  BlendingMode.EXACT_STOP           : StrReplace('EXACT_STOP ({0})','{0}'           , USINT_TO_STRING(Value));
  BlendingMode.DEFINED_VELOCITY     : StrReplace('DEFINED_VELOCITY ({0})','{0}'     , USINT_TO_STRING(Value));
  BlendingMode.CORNER_DISTANCE      : StrReplace('CORNER_DISTANCE ({0})','{0}'      , USINT_TO_STRING(Value));
  BlendingMode.MAX_CORNER_DEVIATION : StrReplace('MAX_CORNER_DEVIATION ({0})','{0}' , USINT_TO_STRING(Value));
  BlendingMode.CORNER_DISTANCE_2R   : StrReplace('CORNER_DISTANCE_2R ({0})','{0}'   , USINT_TO_STRING(Value));
  BlendingMode.RAMP_OVERLAP         : StrReplace('RAMP_OVERLAP ({0})','{0}'         , USINT_TO_STRING(Value));
  BlendingMode.CORNER_DISTANCE_1R   : StrReplace('CORNER_DISTANCE_1R ({0})','{0}'   , USINT_TO_STRING(Value));

END_CASE

END_FUNCTION

// Library/Functions/Convert/TO_STRING/BYTE_TO_STRING_BIN
FUNCTION BYTE_TO_STRING_BIN : STRING
// ------------------------------------------------------------------------- 
//  SRCI Robot Library                                                
// ------------------------------------------------------------------------- 
//                                                                           
//  Object:      BYTE_TO_STRING_BIN                                       
//  Author:      Thorsten Brach                                                
//  Date:        2025-01-20
//
//  Description:                                              
//    Converts a BYTE to a STRING with binary notation  
//                                                                           
//  Copyright: 
//    (C) 2024 Thorsten Brach. All rights reserved                                                                                                                                            
//             Licensed under the LGPL-3.0 license.
//                                                                           
//  Disclaimer:                                                                           
//    This project is provided without any guarantee and can be used for   
//    private and commercial purposes. Any use is at the user’s 
//    own risk and responsibility.
//
// -------------------------------------------------------------------------
VAR_INPUT
 /// Value to convert
 Value : BYTE; 
END_VAR

BYTE_TO_STRING_BIN := '2#';

IF (Value.7)
THEN
  BYTE_TO_STRING_BIN := CONCAT(BYTE_TO_STRING_BIN, '1');
ELSE
  BYTE_TO_STRING_BIN := CONCAT(BYTE_TO_STRING_BIN, '0');
END_IF

IF (Value.6)
THEN
  BYTE_TO_STRING_BIN := CONCAT(BYTE_TO_STRING_BIN, '1');
ELSE
  BYTE_TO_STRING_BIN := CONCAT(BYTE_TO_STRING_BIN, '0');
END_IF

IF (Value.5)
THEN
  BYTE_TO_STRING_BIN := CONCAT(BYTE_TO_STRING_BIN, '1');
ELSE
  BYTE_TO_STRING_BIN := CONCAT(BYTE_TO_STRING_BIN, '0');
END_IF

IF (Value.4)
THEN
  BYTE_TO_STRING_BIN := CONCAT(BYTE_TO_STRING_BIN, '1_');
ELSE
  BYTE_TO_STRING_BIN := CONCAT(BYTE_TO_STRING_BIN, '0_');
END_IF

IF (Value.3)
THEN
  BYTE_TO_STRING_BIN := CONCAT(BYTE_TO_STRING_BIN, '1');
ELSE
  BYTE_TO_STRING_BIN := CONCAT(BYTE_TO_STRING_BIN, '0');
END_IF

IF (Value.2)
THEN
  BYTE_TO_STRING_BIN := CONCAT(BYTE_TO_STRING_BIN, '1');
ELSE
  BYTE_TO_STRING_BIN := CONCAT(BYTE_TO_STRING_BIN, '0');
END_IF

IF (Value.1)
THEN
  BYTE_TO_STRING_BIN := CONCAT(BYTE_TO_STRING_BIN, '1');
ELSE
  BYTE_TO_STRING_BIN := CONCAT(BYTE_TO_STRING_BIN, '0');
END_IF


IF (Value.0)
THEN
  BYTE_TO_STRING_BIN := CONCAT(BYTE_TO_STRING_BIN, '1');
ELSE
  BYTE_TO_STRING_BIN := CONCAT(BYTE_TO_STRING_BIN, '0');
END_IF


BYTE_TO_STRING_BIN := CONCAT(BYTE_TO_STRING_BIN, ' (');
BYTE_TO_STRING_BIN := CONCAT(BYTE_TO_STRING_BIN, WORD_TO_STRING(Value));
BYTE_TO_STRING_BIN := CONCAT(BYTE_TO_STRING_BIN, ')');

END_FUNCTION

// Library/Functions/Convert/TO_STRING/CIRC_MODE_TO_STRING
FUNCTION CIRC_MODE_TO_STRING : STRING
// ------------------------------------------------------------------------- 
//  SRCI Robot Library                                                
// ------------------------------------------------------------------------- 
//                                                                           
//  Object:      CIRC_MODE_TO_STRING                                       
//  Author:      Thorsten Brach                                                
//  Date:        2025-01-30
//
//  Description:                                              
//   
//                                                                           
//  Copyright: 
//    (C) 2025 Thorsten Brach. All rights reserved                                                                                                                                            
//             Licensed under the LGPL-3.0 license.
//                                                                           
//  Disclaimer:                                                                           
//    This project is provided without any guarantee and can be used for   
//    private and commercial purposes. Any use is at the user’s 
//    own risk and responsibility.
//
// -------------------------------------------------------------------------
VAR_INPUT
  /// CircMode
  Value : CircMode;
END_VAR

CASE Value 
OF

  CircMode.BORDER            : StrReplace('BORDER ({0})'            ,'{0}' , SINT_TO_STRING(Value));
  CircMode.CENTER            : StrReplace('CENTER ({0})'            ,'{0}' , SINT_TO_STRING(Value));
  CircMode.CENTER_WITH_ANGLE : StrReplace('CENTER_WITH_ANGLE ({0})' ,'{0}' , SINT_TO_STRING(Value));
  CircMode.RADIUS            : StrReplace('RADIUS ({0})'            ,'{0}' , SINT_TO_STRING(Value));

END_CASE

END_FUNCTION

// Library/Functions/Convert/TO_STRING/CIRC_PLANE_TO_STRING
FUNCTION CIRC_PLANE_TO_STRING : STRING
// ------------------------------------------------------------------------- 
//  SRCI Robot Library                                                
// ------------------------------------------------------------------------- 
//                                                                           
//  Object:      CIRC_PLANE_TO_STRING                                       
//  Author:      Thorsten Brach                                                
//  Date:        2025-01-30
//
//  Description:                                              
//   
//                                                                           
//  Copyright: 
//    (C) 2025 Thorsten Brach. All rights reserved                                                                                                                                            
//             Licensed under the LGPL-3.0 license.
//                                                                           
//  Disclaimer:                                                                           
//    This project is provided without any guarantee and can be used for   
//    private and commercial purposes. Any use is at the user’s 
//    own risk and responsibility.
//
// -------------------------------------------------------------------------
VAR_INPUT
  /// CircPlane
  Value : CircPlane;
END_VAR

CASE Value 
OF

  CircPlane.XZ_PLANE : StrReplace('XZ_PLANE ({0})' ,'{0}' , SINT_TO_STRING(Value));
  CircPlane.YZ_PLANE : StrReplace('YZ_PLANE ({0})' ,'{0}' , SINT_TO_STRING(Value));
  CircPlane.XY_PLANE : StrReplace('XY_PLANE ({0})' ,'{0}' , SINT_TO_STRING(Value));

END_CASE

END_FUNCTION

// Library/Functions/Convert/TO_STRING/CMD_MESSAGE_STATE_TO_STRING
FUNCTION CMD_MESSAGE_STATE_TO_STRING : STRING
// ------------------------------------------------------------------------- 
//  SRCI Robot Library                                                
// ------------------------------------------------------------------------- 
//                                                                           
//  Object:      CMD_MESSAGE_STATE_TO_STRING                                       
//  Author:      Thorsten Brach                                                
//  Date:        2024-11-16
//
//  Description:                                              
//   
//                                                                           
//  Copyright: 
//    (C) 2024 Thorsten Brach. All rights reserved                                                                                                                                            
//             Licensed under the LGPL-3.0 license.
//                                                                           
//  Disclaimer:                                                                           
//    This project is provided without any guarantee and can be used for   
//    private and commercial purposes. Any use is at the user’s 
//    own risk and responsibility.
//
// -------------------------------------------------------------------------
VAR_INPUT
  /// Command message state
  Value : CmdMessageState;
END_VAR

CASE Value
OF
  CmdMessageState.EMPTY               : CMD_MESSAGE_STATE_TO_STRING := StrReplace('EMPTY ({0})'              ,'{0}', USINT_TO_STRING(Value));
  CmdMessageState.CREATED             : CMD_MESSAGE_STATE_TO_STRING := StrReplace('CREATED ({0})'            ,'{0}', USINT_TO_STRING(Value));
  CmdMessageState.BUFFERED            : CMD_MESSAGE_STATE_TO_STRING := StrReplace('BUFFERED ({0})'           ,'{0}', USINT_TO_STRING(Value));
  CmdMessageState.BUFFERED_IN_PLANNER : CMD_MESSAGE_STATE_TO_STRING := StrReplace('BUFFERED_IN_PLANNER ({0})','{0}', USINT_TO_STRING(Value));
  CmdMessageState.ACTIVE              : CMD_MESSAGE_STATE_TO_STRING := StrReplace('ACTIVE ({0})'             ,'{0}', USINT_TO_STRING(Value));
  CmdMessageState.INTERRUPTED         : CMD_MESSAGE_STATE_TO_STRING := StrReplace('INTERRUPTED ({0})'        ,'{0}', USINT_TO_STRING(Value));
  CmdMessageState.ABORT_REQUEST       : CMD_MESSAGE_STATE_TO_STRING := StrReplace('ABORT_REQUEST ({0})'      ,'{0}', USINT_TO_STRING(Value));
  CmdMessageState.DONE                : CMD_MESSAGE_STATE_TO_STRING := StrReplace('DONE ({0})'               ,'{0}', USINT_TO_STRING(Value));
  CmdMessageState.ABORTED             : CMD_MESSAGE_STATE_TO_STRING := StrReplace('ABORTED ({0})'            ,'{0}', USINT_TO_STRING(Value));
  CmdMessageState.ERROR               : CMD_MESSAGE_STATE_TO_STRING := StrReplace('ERROR ({0})'              ,'{0}', USINT_TO_STRING(Value));
ELSE
  CMD_MESSAGE_STATE_TO_STRING := CONCAT('CmdMessageStateToString-Function: Error -> no parsing for value ', USINT_TO_STRING(Value));
END_CASE

END_FUNCTION

// Library/Functions/Convert/TO_STRING/CMD_TYPE_TO_STRING
FUNCTION CMD_TYPE_TO_STRING : String
// ------------------------------------------------------------------------- 
//  SRCI Robot Library                                                
// ------------------------------------------------------------------------- 
//                                                                           
//  Object:      CMD_TYPE_TO_STRING                                       
//  Author:      Thorsten Brach                                                
//  Date:        2024-11-16
//
//  Description:                                              
//   
//                                                                           
//  Copyright: 
//    (C) 2024 Thorsten Brach. All rights reserved                                                                                                                                            
//             Licensed under the LGPL-3.0 license.
//                                                                           
//  Disclaimer:                                                                           
//    This project is provided without any guarantee and can be used for   
//    private and commercial purposes. Any use is at the user’s 
//    own risk and responsibility.
//
// -------------------------------------------------------------------------
VAR_INPUT
  /// command type
  Value : CmdType;
END_VAR

CASE Value 
OF
  CmdType.RobotTask                   : CMD_TYPE_TO_STRING := StrReplace('RobotTask ({0})','{0}'                  , UINT_TO_STRING(CmdType.RobotTask));   

  CmdType.ReadRobotData               : CMD_TYPE_TO_STRING := StrReplace('ReadRobotData ({0})','{0}'              , UINT_TO_STRING(CmdType.ReadRobotData));

  CmdType.EnableRobot                 : CMD_TYPE_TO_STRING := StrReplace('EnableRobot ({0})','{0}'                , UINT_TO_STRING(CmdType.EnableRobot));  

  CmdType.GroupReset                  : CMD_TYPE_TO_STRING := StrReplace('GroupReset ({0})','{0}'                 , UINT_TO_STRING(CmdType.GroupReset));  

  CmdType.ReadActualPosition          : CMD_TYPE_TO_STRING := StrReplace('ReadActualPosition ({0})','{0}'         , UINT_TO_STRING(CmdType.ReadActualPosition));

  CmdType.ReadActualPositionCyclic    : CMD_TYPE_TO_STRING := StrReplace('ReadActualPositionCyclic ({0})','{0}'   , UINT_TO_STRING(CmdType.ReadActualPositionCyclic));  

  CmdType.ReadDHParameter             : CMD_TYPE_TO_STRING := StrReplace('ReadDHParameter ({0})','{0}'            , UINT_TO_STRING(CmdType.ReadDHParameter));  

  CmdType.RestartController           : CMD_TYPE_TO_STRING := StrReplace('RestartController ({0})','{0}'          , UINT_TO_STRING(CmdType.RestartController));  

  CmdType.ReadActualTCPVelocity       : CMD_TYPE_TO_STRING := StrReplace('ReadActualTCPVelocity ({0})','{0}'      , UINT_TO_STRING(CmdType.ReadActualTCPVelocity));  

  CmdType.UserLogin                   : CMD_TYPE_TO_STRING := StrReplace('UserLogin ({0})','{0}'                  , UINT_TO_STRING(CmdType.UserLogin));

  CmdType.SwitchLanguage              : CMD_TYPE_TO_STRING := StrReplace('SwitchLanguage ({0})','{0}'             , UINT_TO_STRING(CmdType.SwitchLanguage));

  CmdType.ExchangeConfiguration       : CMD_TYPE_TO_STRING := StrReplace('ExchangeConfiguration ({0})','{0}'      , UINT_TO_STRING(CmdType.ExchangeConfiguration));

  CmdType.SetSequence                 : CMD_TYPE_TO_STRING := StrReplace('SetSequence ({0})','{0}'                , UINT_TO_STRING(CmdType.SetSequence));

  CmdType.ChangeSpeedOverride         : CMD_TYPE_TO_STRING := StrReplace('ChangeSpeedOverride ({0})','{0}'        , UINT_TO_STRING(CmdType.ChangeSpeedOverride));

  CmdType.ReadMessages                : CMD_TYPE_TO_STRING := StrReplace('ReadMessages ({0})','{0}'               , UINT_TO_STRING(CmdType.ReadMessages));

  CmdType.ReadRobotReferenceDynamics  : CMD_TYPE_TO_STRING := StrReplace('ReadRobotReferenceDynamics ({0})','{0}' , UINT_TO_STRING(CmdType.ReadRobotReferenceDynamics));  

  CmdType.WriteFrameData              : CMD_TYPE_TO_STRING := StrReplace('WriteFrameData ({0})','{0}'             , UINT_TO_STRING(CmdType.WriteFrameData));

  CmdType.WriteToolData               : CMD_TYPE_TO_STRING := StrReplace('WriteToolData ({0})','{0}'              , UINT_TO_STRING(CmdType.WriteToolData));

  CmdType.WriteLoadData               : CMD_TYPE_TO_STRING := StrReplace('WriteLoadData ({0})','{0}'              , UINT_TO_STRING(CmdType.WriteLoadData));

  CmdType.WriteRobotReferenceDynamics : CMD_TYPE_TO_STRING := StrReplace('WriteRobotReferenceDynamics ({0})','{0}', UINT_TO_STRING(CmdType.WriteRobotReferenceDynamics));

  CmdType.WriteRobotDefaultDynamics   : CMD_TYPE_TO_STRING := StrReplace('WriteRobotDefaultDynamics ({0})'  ,'{0}', UINT_TO_STRING(CmdType.WriteRobotDefaultDynamics));

  CmdType.ReadRobotDefaultDynamics    : CMD_TYPE_TO_STRING := StrReplace('ReadRobotDefaultDynamics ({0})'   ,'{0}', UINT_TO_STRING(CmdType.ReadRobotDefaultDynamics));

  CmdType.ReadFrameData               : CMD_TYPE_TO_STRING := StrReplace('ReadFrameData ({0})'              ,'{0}', UINT_TO_STRING(CmdType.ReadFrameData)); 

  CmdType.ReadToolData                : CMD_TYPE_TO_STRING := StrReplace('ReadToolData ({0})','{0}'               , UINT_TO_STRING(CmdType.ReadToolData));

  CmdType.ReadLoadData                : CMD_TYPE_TO_STRING := StrReplace('ReadLoadData ({0})','{0}'               , UINT_TO_STRING(CmdType.ReadLoadData));

  CmdType.ReadRobotSWLimits           : CMD_TYPE_TO_STRING := StrReplace('ReadRobotSWLimits ({0})','{0}'          , UINT_TO_STRING(CmdType.ReadRobotSWLimits));

  CmdType.WriteRobotSWLimits          : CMD_TYPE_TO_STRING := StrReplace('WriteRobotSWLimits ({0})','{0}'         , UINT_TO_STRING(CmdType.WriteRobotSWLimits));

  CmdType.SetOperationMode            : CMD_TYPE_TO_STRING := StrReplace('SetOperationMode ({0})','{0}'           , UINT_TO_STRING(CmdType.SetOperationMode));

  CmdType.ReadWorkArea                : CMD_TYPE_TO_STRING := StrReplace('ReadWorkArea ({0})','{0}'               , UINT_TO_STRING(CmdType.ReadWorkArea));

  CmdType.WriteWorkArea               : CMD_TYPE_TO_STRING := StrReplace('WriteWorkArea ({0})','{0}'              , UINT_TO_STRING(CmdType.WriteWorkArea));

  CmdType.ActivateWorkArea            : CMD_TYPE_TO_STRING := StrReplace('ActivateWorkArea ({0})','{0}'           , UINT_TO_STRING(CmdType.ActivateWorkArea));

  CmdType.MonitorWorkArea             : CMD_TYPE_TO_STRING := StrReplace('MonitorWorkArea ({0})','{0}'            , UINT_TO_STRING(CmdType.MonitorWorkArea));

  CmdType.GroupJog                    : CMD_TYPE_TO_STRING := StrReplace('GroupJog ({0})','{0}'                   , UINT_TO_STRING(CmdType.GroupJog));

  CmdType.MoveLinearAbsolute          : CMD_TYPE_TO_STRING := StrReplace('MoveLinearAbsolute ({0})','{0}'         , UINT_TO_STRING(CmdType.MoveLinearAbsolute));

  CmdType.MoveDirectAbsolute          : CMD_TYPE_TO_STRING := StrReplace('MoveDirectAbsolute ({0})','{0}'         , UINT_TO_STRING(CmdType.MoveDirectAbsolute));

  CmdType.MoveAxesAbsolute            : CMD_TYPE_TO_STRING := StrReplace('MoveAxesAbsolute ({0})','{0}'           , UINT_TO_STRING(CmdType.MoveAxesAbsolute));

  CmdType.GroupStop                   : CMD_TYPE_TO_STRING := StrReplace('GroupStop ({0})','{0}'                  , UINT_TO_STRING(CmdType.GroupStop));

  CmdType.GroupInterrupt              : CMD_TYPE_TO_STRING := StrReplace('GroupInterrupt ({0})','{0}'             , UINT_TO_STRING(CmdType.GroupInterrupt));

  CmdType.GroupContinue               : CMD_TYPE_TO_STRING := StrReplace('GroupContinue ({0})','{0}'              , UINT_TO_STRING(CmdType.GroupContinue));

  CmdType.MoveLinearRelative          : CMD_TYPE_TO_STRING := StrReplace('MoveLinearRelative ({0})','{0}'         , UINT_TO_STRING(CmdType.MoveLinearRelative));

  CmdType.MoveDirectRelative          : CMD_TYPE_TO_STRING := StrReplace('MoveDirectRelative ({0})','{0}'         , UINT_TO_STRING(CmdType.MoveDirectRelative));

  CmdType.MoveAxesRelative            : CMD_TYPE_TO_STRING := StrReplace('MoveAxesRelative ({0})','{0}'           , UINT_TO_STRING(CmdType.MoveAxesRelative));

  CmdType.ReturnToPrimary             : CMD_TYPE_TO_STRING := StrReplace('ReturnToPrimary ({0})','{0}'            , UINT_TO_STRING(CmdType.ReturnToPrimary));

  CmdType.MoveCircularAbsolute        : CMD_TYPE_TO_STRING := StrReplace('MoveCircularAbsolute ({0})','{0}'       , UINT_TO_STRING(CmdType.MoveCircularAbsolute));

  CmdType.MoveCircularRelative        : CMD_TYPE_TO_STRING := StrReplace('MoveCircularRelative ({0})','{0}'       , UINT_TO_STRING(CmdType.MoveCircularRelative));

  CmdType.MoveLinearOffset            : CMD_TYPE_TO_STRING := StrReplace('MoveLinearOffset ({0})','{0}'           , UINT_TO_STRING(CmdType.MoveLinearOffset));

  CmdType.MoveDirectOffset            : CMD_TYPE_TO_STRING := StrReplace('MoveDirectOffset ({0})','{0}'           , UINT_TO_STRING(CmdType.MoveDirectOffset));

  CmdType.WaitTime                    : CMD_TYPE_TO_STRING := StrReplace('WaitTime ({0})','{0}'                   , UINT_TO_STRING(CmdType.WaitTime));

  CmdType.MoveApproachLinear          : CMD_TYPE_TO_STRING := StrReplace('MoveApproachLinear ({0})','{0}'         , UINT_TO_STRING(CmdType.MoveApproachLinear));

  CmdType.MoveDepartLinear            : CMD_TYPE_TO_STRING := StrReplace('MoveDepartLinear ({0})','{0}'           , UINT_TO_STRING(CmdType.MoveDepartLinear));

  CmdType.MoveApproachDirect          : CMD_TYPE_TO_STRING := StrReplace('MoveApproachDirect ({0})','{0}'         , UINT_TO_STRING(CmdType.MoveApproachDirect));

  CmdType.MoveDepartDirect            : CMD_TYPE_TO_STRING := StrReplace('MoveDepartDirect ({0})','{0}'           , UINT_TO_STRING(CmdType.MoveDepartDirect));

  CmdType.SearchHardstop              : CMD_TYPE_TO_STRING := StrReplace('SearchHardstop ({0})','{0}'             , UINT_TO_STRING(CmdType.SearchHardstop));

  CmdType.SearchHardstopJ             : CMD_TYPE_TO_STRING := StrReplace('SearchHardstopJ ({0})','{0}'            , UINT_TO_STRING(CmdType.SearchHardstopJ));

  CmdType.MovePickPlaceLinear         : CMD_TYPE_TO_STRING := StrReplace('MovePickPlaceLinear ({0})','{0}'        , UINT_TO_STRING(CmdType.MovePickPlaceLinear));

  CmdType.MovePickPlaceDirect         : CMD_TYPE_TO_STRING := StrReplace('MovePickPlaceDirect ({0})','{0}'        , UINT_TO_STRING(CmdType.MovePickPlaceDirect));  

  CmdType.ActivateConveyorTracking    : CMD_TYPE_TO_STRING := StrReplace('ActivateConveyorTracking ({0})','{0}'   , UINT_TO_STRING(CmdType.ActivateConveyorTracking));

  CmdType.RedefineTrackingPos         : CMD_TYPE_TO_STRING := StrReplace('RedefineTrackingPos ({0})','{0}'        , UINT_TO_STRING(CmdType.RedefineTrackingPos));

  CmdType.SyncToConveyor              : CMD_TYPE_TO_STRING := StrReplace('SyncToConveyor ({0})','{0}'             , UINT_TO_STRING(CmdType.SyncToConveyor));

  CmdType.ConfigureConveyor           : CMD_TYPE_TO_STRING := StrReplace('ConfigureConveyor ({0})','{0}'          , UINT_TO_STRING(CmdType.ConfigureConveyor));

  CmdType.MoveSuperImposed            : CMD_TYPE_TO_STRING := StrReplace('MoveSuperImposed ({0})','{0}'           , UINT_TO_STRING(CmdType.MoveSuperImposed));

  CmdType.MoveSuperImposedDynamic     : CMD_TYPE_TO_STRING := StrReplace('MoveSuperImposedDynamic ({0})','{0}'    , UINT_TO_STRING(CmdType.MoveSuperImposedDynamic));

  CmdType.ReadDigitalInputs           : CMD_TYPE_TO_STRING := StrReplace('ReadDigitalInputs ({0})','{0}'          , UINT_TO_STRING(CmdType.ReadDigitalInputs));

  CmdType.ReadDigitalOutputs          : CMD_TYPE_TO_STRING := StrReplace('ReadDigitalOutputs ({0})','{0}'         , UINT_TO_STRING(CmdType.ReadDigitalOutputs));

  CmdType.WriteDigitalOutputs         : CMD_TYPE_TO_STRING := StrReplace('WriteDigitalOutputs ({0})','{0}'        , UINT_TO_STRING(CmdType.WriteDigitalOutputs));

  CmdType.ReadIntegers                : CMD_TYPE_TO_STRING := StrReplace('ReadIntegers ({0})','{0}'               , UINT_TO_STRING(CmdType.ReadIntegers));

  CmdType.ReadReals                   : CMD_TYPE_TO_STRING := StrReplace('ReadReals ({0})','{0}'                  , UINT_TO_STRING(CmdType.ReadReals));

  CmdType.WriteIntegers               : CMD_TYPE_TO_STRING := StrReplace('WriteIntegers ({0})','{0}'              , UINT_TO_STRING(CmdType.WriteIntegers));

  CmdType.WriteReals                  : CMD_TYPE_TO_STRING := StrReplace('WriteReals ({0})','{0}'                 , UINT_TO_STRING(CmdType.WriteReals));

  CmdType.MoveLinearCam               : CMD_TYPE_TO_STRING := StrReplace('MoveLinearCam ({0})','{0}'              , UINT_TO_STRING(CmdType.MoveLinearCam));

  CmdType.MoveDirectCam               : CMD_TYPE_TO_STRING := StrReplace('MoveDirectCam ({0})','{0}'              , UINT_TO_STRING(CmdType.MoveDirectCam));

  CmdType.MoveCircularCam             : CMD_TYPE_TO_STRING := StrReplace('MoveCircularCam ({0})','{0}'            , UINT_TO_STRING(CmdType.MoveCircularCam));

  CmdType.ReadAnalogInput             : CMD_TYPE_TO_STRING := StrReplace('ReadAnalogInput ({0})','{0}'            , UINT_TO_STRING(CmdType.ReadAnalogInput));

  CmdType.ReadAnalogOutput            : CMD_TYPE_TO_STRING := StrReplace('ReadAnalogOutput ({0})','{0}'           , UINT_TO_STRING(CmdType.ReadAnalogOutput));

  CmdType.WriteAnalogOutput           : CMD_TYPE_TO_STRING := StrReplace('WriteAnalogOutput ({0})','{0}'          , UINT_TO_STRING(CmdType.WriteAnalogOutput));

  CmdType.MeasuringInput              : CMD_TYPE_TO_STRING := StrReplace('MeasuringInput ({0})','{0}'             , UINT_TO_STRING(CmdType.MeasuringInput));

  CmdType.AbortMeasuringInput         : CMD_TYPE_TO_STRING := StrReplace('AbortMeasuringInput ({0})','{0}'        , UINT_TO_STRING(CmdType.AbortMeasuringInput));

  CmdType.SetTriggerRegister          : CMD_TYPE_TO_STRING := StrReplace('SetTriggerRegister ({0})','{0}'         , UINT_TO_STRING(CmdType.SetTriggerRegister));

  CmdType.SetTriggerLimit             : CMD_TYPE_TO_STRING := StrReplace('SetTriggerLimit ({0})','{0}'            , UINT_TO_STRING(CmdType.SetTriggerLimit));

  CmdType.SetTriggerUser              : CMD_TYPE_TO_STRING := StrReplace('SetTriggerUser ({0})','{0}'             , UINT_TO_STRING(CmdType.SetTriggerUser));

  CmdType.SetTriggerError             : CMD_TYPE_TO_STRING := StrReplace('SetTriggerError ({0})','{0}'            , UINT_TO_STRING(CmdType.SetTriggerError));

  CmdType.ReactAtTrigger              : CMD_TYPE_TO_STRING := StrReplace('ReactAtTrigger ({0})','{0}'             , UINT_TO_STRING(CmdType.ReactAtTrigger));

  CmdType.WaitForTrigger              : CMD_TYPE_TO_STRING := StrReplace('WaitForTrigger ({0})','{0}'             , UINT_TO_STRING(CmdType.WaitForTrigger));

  CmdType.ReadSystemVariable          : CMD_TYPE_TO_STRING := StrReplace('ReadSystemVariable ({0})','{0}'         , UINT_TO_STRING(CmdType.ReadSystemVariable));

  CmdType.WriteSystemVariable         : CMD_TYPE_TO_STRING := StrReplace('WriteSystemVariable ({0})','{0}'        , UINT_TO_STRING(CmdType.WriteSystemVariable));

  CmdType.CalculateForwardKinematic   : CMD_TYPE_TO_STRING := StrReplace('CalculateForwardKinematic ({0})','{0}'  , UINT_TO_STRING(CmdType.CalculateForwardKinematic));

  CmdType.CalculateInverseKinematic   : CMD_TYPE_TO_STRING := StrReplace('CalculateInverseKinematic ({0})','{0}'  , UINT_TO_STRING(CmdType.CalculateInverseKinematic));

  CmdType.CalculateCartesianPosition  : CMD_TYPE_TO_STRING := StrReplace('CalculateCartesianPosition ({0})','{0}' , UINT_TO_STRING(CmdType.CalculateCartesianPosition));

  CmdType.CalculateTool               : CMD_TYPE_TO_STRING := StrReplace('CalculateTool ({0})','{0}'              , UINT_TO_STRING(CmdType.CalculateTool));

  CmdType.CalculateFrame              : CMD_TYPE_TO_STRING := StrReplace('CalculateFrame ({0})','{0}'             , UINT_TO_STRING(CmdType.CalculateFrame));

  CmdType.ActivateNextCommand         : CMD_TYPE_TO_STRING := StrReplace('ActivateNextCommand ({0})','{0}'        , UINT_TO_STRING(CmdType.ActivateNextCommand));

  CmdType.ShiftPosition               : CMD_TYPE_TO_STRING := StrReplace('ShiftPosition ({0})','{0}'              , UINT_TO_STRING(CmdType.ShiftPosition));

  CmdType.SetTriggerMotion            : CMD_TYPE_TO_STRING := StrReplace('SetTriggerMotion ({0})','{0}'           , UINT_TO_STRING(CmdType.SetTriggerMotion));

  CmdType.OpenBrake                   : CMD_TYPE_TO_STRING := StrReplace('OpenBrake ({0})','{0}'                  , UINT_TO_STRING(CmdType.OpenBrake));

  CmdType.CallSubprogram              : CMD_TYPE_TO_STRING := StrReplace('CallSubprogram ({0})','{0}'             , UINT_TO_STRING(CmdType.CallSubprogram));

  CmdType.WriteCallSubprogramCyclic   : CMD_TYPE_TO_STRING := StrReplace('WriteCallSubprogramCyclic ({0})','{0}'  , UINT_TO_STRING(CmdType.WriteCallSubprogramCyclic));

  CmdType.ReadCallSubprogramCyclic    : CMD_TYPE_TO_STRING := StrReplace('ReadCallSubprogramCyclic ({0})','{0}'   , UINT_TO_STRING(CmdType.ReadCallSubprogramCyclic));

  CmdType.StopSubprogram              : CMD_TYPE_TO_STRING := StrReplace('StopSubprogram ({0})','{0}'             , UINT_TO_STRING(CmdType.StopSubprogram));

  CmdType.PathAccuracyMode            : CMD_TYPE_TO_STRING := StrReplace('PathAccuracyMode ({0})','{0}'           , UINT_TO_STRING(CmdType.PathAccuracyMode));

  CmdType.AvoidSingularity            : CMD_TYPE_TO_STRING := StrReplace('AvoidSingularity ({0})','{0}'           , UINT_TO_STRING(CmdType.AvoidSingularity));

  CmdType.ForceControl                : CMD_TYPE_TO_STRING := StrReplace('ForceControl ({0})','{0}'               , UINT_TO_STRING(CmdType.ForceControl));

  CmdType.ForceLimit                  : CMD_TYPE_TO_STRING := StrReplace('ForceLimit ({0})','{0}'                 , UINT_TO_STRING(CmdType.ForceLimit));

  CmdType.ReadActualForce             : CMD_TYPE_TO_STRING := StrReplace('ReadActualForce ({0})','{0}'            , UINT_TO_STRING(CmdType.ReadActualForce));

  CmdType.BrakeTest                   : CMD_TYPE_TO_STRING := StrReplace('BrakeTest ({0})','{0}'                  , UINT_TO_STRING(CmdType.BrakeTest));

  CmdType.SoftSwitchTCP               : CMD_TYPE_TO_STRING := StrReplace('SoftSwitchTCP ({0})','{0}'              , UINT_TO_STRING(CmdType.SoftSwitchTCP));

  CmdType.CreateSpline                : CMD_TYPE_TO_STRING := StrReplace('CreateSpline ({0})','{0}'               , UINT_TO_STRING(CmdType.CreateSpline));

  CmdType.DeleteSpline                : CMD_TYPE_TO_STRING := StrReplace('DeleteSpline ({0})','{0}'               , UINT_TO_STRING(CmdType.DeleteSpline));

  CmdType.MoveSpline                  : CMD_TYPE_TO_STRING := StrReplace('MoveSpline ({0})','{0}'                 , UINT_TO_STRING(CmdType.MoveSpline));

  CmdType.DynamicSpline               : CMD_TYPE_TO_STRING := StrReplace('DynamicSpline ({0})','{0}'              , UINT_TO_STRING(CmdType.DynamicSpline));

  CmdType.LoadMeasurementAutomatic    : CMD_TYPE_TO_STRING := StrReplace('LoadMeasurementAutomatic ({0})','{0}'   , UINT_TO_STRING(CmdType.LoadMeasurementAutomatic));

  CmdType.LoadMeasurementSequential   : CMD_TYPE_TO_STRING := StrReplace('LoadMeasurementSequential ({0})','{0}'  , UINT_TO_STRING(CmdType.LoadMeasurementSequential));

  CmdType.CollisionDetection          : CMD_TYPE_TO_STRING := StrReplace('CollisionDetection ({0})','{0}'         , UINT_TO_STRING(CmdType.CollisionDetection));

  CmdType.FreeDrive                   : CMD_TYPE_TO_STRING := StrReplace('FreeDrive ({0})','{0}'                  , UINT_TO_STRING(CmdType.FreeDrive)); 

  CmdType.UnitMeasurement             : CMD_TYPE_TO_STRING := StrReplace('UnitMeasurement ({0})','{0}'            , UINT_TO_STRING(CmdType.UnitMeasurement));

ELSE
  CMD_TYPE_TO_STRING := CONCAT('CmdTypeToString-Function: Error -> no parsing for value',UINT_TO_STRING(Value));
END_CASE

END_FUNCTION

// Library/Functions/Convert/TO_STRING/COLLISION_REACTION_MODE_TO_STRING
FUNCTION COLLISION_REACTION_MODE_TO_STRING : STRING
// ------------------------------------------------------------------------- 
//  SRCI Robot Library                                                
// ------------------------------------------------------------------------- 
//                                                                           
//  Object:      COLLISION_REACTION_MODE_TO_STRING                                       
//  Author:      Thorsten Brach                                                
//  Date:        2025-01-24
//
//  Description:                                              
//   
//                                                                           
//  Copyright: 
//    (C) 2025 Thorsten Brach. All rights reserved                                                                                                                                            
//             Licensed under the LGPL-3.0 license.
//                                                                           
//  Disclaimer:                                                                           
//    This project is provided without any guarantee and can be used for   
//    private and commercial purposes. Any use is at the user’s 
//    own risk and responsibility.
//
// -------------------------------------------------------------------------
VAR_INPUT
  /// CollisionReactionMode
  Value : CollisionReactionMode;
END_VAR

CASE Value 
OF

  CollisionReactionMode.REVERSED_MOVEMENT : StrReplace('REVERSED_MOVEMENT ({0})','{0}' , USINT_TO_STRING(Value));
  CollisionReactionMode.STANDING_STILL    : StrReplace('STANDING_STILL ({0})'   ,'{0}' , USINT_TO_STRING(Value));

END_CASE

END_FUNCTION

// Library/Functions/Convert/TO_STRING/CONNECTION_MODE_TO_STRING
FUNCTION CONNECTION_MODE_TO_STRING : STRING
// ------------------------------------------------------------------------- 
//  SRCI Robot Library                                                
// ------------------------------------------------------------------------- 
//                                                                           
//  Object:      CONNECTION_MODE_TO_STRING                                       
//  Author:      Thorsten Brach                                                
//  Date:        2025-02-01
//
//  Description:                                              
//   
//                                                                           
//  Copyright: 
//    (C) 2025 Thorsten Brach. All rights reserved                                                                                                                                            
//             Licensed under the LGPL-3.0 license.
//                                                                           
//  Disclaimer:                                                                           
//    This project is provided without any guarantee and can be used for   
//    private and commercial purposes. Any use is at the user’s 
//    own risk and responsibility.
//
// -------------------------------------------------------------------------
VAR_INPUT
  /// ConnectionMode
  Value : ConnectionMode;
END_VAR

CASE Value 
OF

  ConnectionMode.RC_CONNECTED  : StrReplace('RC_CONNECTED ({0})'  ,'{0}' , SINT_TO_STRING(Value));
  ConnectionMode.PLC_CONNECTED : StrReplace('PLC_CONNECTED ({0})' ,'{0}' , SINT_TO_STRING(Value));

END_CASE

END_FUNCTION

// Library/Functions/Convert/TO_STRING/CONVEYOR_TYPE_TO_STRING
FUNCTION CONVEYOR_TYPE_TO_STRING : STRING
// ------------------------------------------------------------------------- 
//  SRCI Robot Library                                                
// ------------------------------------------------------------------------- 
//                                                                           
//  Object:      CONVEYOR_TYPE_TO_STRING                                       
//  Author:      Thorsten Brach                                                
//  Date:        2025-02-01
//
//  Description:                                              
//   
//                                                                           
//  Copyright: 
//    (C) 2025 Thorsten Brach. All rights reserved                                                                                                                                            
//             Licensed under the LGPL-3.0 license.
//                                                                           
//  Disclaimer:                                                                           
//    This project is provided without any guarantee and can be used for   
//    private and commercial purposes. Any use is at the user’s 
//    own risk and responsibility.
//
// -------------------------------------------------------------------------
VAR_INPUT
  /// ConveyorType
  Value : ConveyorType;
END_VAR

CASE Value 
OF

  ConveyorType.LINEAR_CONVEYOR_TRACKING   : StrReplace('LINEAR_CONVEYOR_TRACKING ({0})'   ,'{0}' , USINT_TO_STRING(Value));
  ConveyorType.CIRCULAR_CONVEYOR_TRACKING : StrReplace('CIRCULAR_CONVEYOR_TRACKING ({0})' ,'{0}' , USINT_TO_STRING(Value));
  
END_CASE

END_FUNCTION

// Library/Functions/Convert/TO_STRING/DATA_ENABLE_SYNC_TO_STRING
FUNCTION DATA_ENABLE_SYNC_TO_STRING : STRING
// ------------------------------------------------------------------------- 
//  SRCI Robot Library                                                
// ------------------------------------------------------------------------- 
//                                                                           
//  Object:      DATA_ENABLE_SYNC_TO_STRING                                       
//  Author:      Thorsten Brach                                                
//  Date:        2025-01-24
//
//  Description:                                              
//   
//                                                                           
//  Copyright: 
//    (C) 2025 Thorsten Brach. All rights reserved                                                                                                                                            
//             Licensed under the LGPL-3.0 license.
//                                                                           
//  Disclaimer:                                                                           
//    This project is provided without any guarantee and can be used for   
//    private and commercial purposes. Any use is at the user’s 
//    own risk and responsibility.
//
// -------------------------------------------------------------------------
VAR_INPUT
  /// DataEnableSync
  Value : DataEnableSync;
END_VAR

VAR
  /// temporary byte
 _tmpByte : BYTE;
END_VAR

_tmpByte.0 := Value.EnableSyncTool;
_tmpByte.1 := Value.EnableSyncFrame;
_tmpByte.2 := Value.EnableSyncLoad;
_tmpByte.3 := Value.EnableSyncWorkArea;
_tmpByte.4 := Value.EnableSyncSWLimits;
_tmpByte.5 := Value.EnableSyncDefaultDynamics;
_tmpByte.6 := Value.EnableSyncReferenceDynamics;
_tmpByte.7 := Value.AllowDynamicBlending;

DATA_ENABLE_SYNC_TO_STRING := BYTE_TO_STRING_BIN(_tmpByte);

END_FUNCTION

// Library/Functions/Convert/TO_STRING/DATA_IN_SYNC_TO_STRING
FUNCTION DATA_IN_SYNC_TO_STRING : STRING
// ------------------------------------------------------------------------- 
//  SRCI Robot Library                                                
// ------------------------------------------------------------------------- 
//                                                                           
//  Object:      DATA_IN_SYNC_TO_STRING                                       
//  Author:      Thorsten Brach                                                
//  Date:        2025-01-24
//
//  Description:                                              
//   
//                                                                           
//  Copyright: 
//    (C) 2025 Thorsten Brach. All rights reserved                                                                                                                                            
//             Licensed under the LGPL-3.0 license.
//                                                                           
//  Disclaimer:                                                                           
//    This project is provided without any guarantee and can be used for   
//    private and commercial purposes. Any use is at the user’s 
//    own risk and responsibility.
//
// -------------------------------------------------------------------------
VAR_INPUT
  /// DataInSync
  Value : DataInSync;
END_VAR

VAR
  /// temporary byte
 _tmpByte : BYTE;
END_VAR

_tmpByte.0 := Value.ToolsInSync;
_tmpByte.1 := Value.FramesInSync;
_tmpByte.2 := Value.LoadsInSync;
_tmpByte.3 := Value.WorkAreasInSync;
_tmpByte.4 := Value.SoftwareLimitsInSync;
_tmpByte.5 := Value.DefaultDynamicsInSync;
_tmpByte.6 := Value.ReferenceDynamicsInSync;
_tmpByte.7 := FALSE;

DATA_IN_SYNC_TO_STRING := BYTE_TO_STRING_BIN(_tmpByte);

END_FUNCTION

// Library/Functions/Convert/TO_STRING/DEFINITION_MODE_TO_STRING
FUNCTION DEFINITION_MODE_TO_STRING : STRING
// ------------------------------------------------------------------------- 
//  SRCI Robot Library                                                
// ------------------------------------------------------------------------- 
//                                                                           
//  Object:      DEFINITION_MODE_TO_STRING                                       
//  Author:      Thorsten Brach                                                
//  Date:        2025-02-01
//
//  Description:                                              
//   
//                                                                           
//  Copyright: 
//    (C) 2025 Thorsten Brach. All rights reserved                                                                                                                                            
//             Licensed under the LGPL-3.0 license.
//                                                                           
//  Disclaimer:                                                                           
//    This project is provided without any guarantee and can be used for   
//    private and commercial purposes. Any use is at the user’s 
//    own risk and responsibility.
//
// -------------------------------------------------------------------------
VAR_INPUT
  /// DefinitionMode
  Value : DefinitionMode;
END_VAR

CASE Value 
OF

  DefinitionMode.CENTER : StrReplace('CENTER ({0})','{0}' , USINT_TO_STRING(Value));
  DefinitionMode.FACE   : StrReplace('FACE ({0})'  ,'{0}' , USINT_TO_STRING(Value));

END_CASE

END_FUNCTION

// Library/Functions/Convert/TO_STRING/DETECTION_MODE_TO_STRING
FUNCTION DETECTION_MODE_TO_STRING : STRING
// ------------------------------------------------------------------------- 
//  SRCI Robot Library                                                
// ------------------------------------------------------------------------- 
//                                                                           
//  Object:      DETECTION_MODE_TO_STRING                                       
//  Author:      Thorsten Brach                                                
//  Date:        2025-02-01
//
//  Description:                                              
//   
//                                                                           
//  Copyright: 
//    (C) 2025 Thorsten Brach. All rights reserved                                                                                                                                            
//             Licensed under the LGPL-3.0 license.
//                                                                           
//  Disclaimer:                                                                           
//    This project is provided without any guarantee and can be used for   
//    private and commercial purposes. Any use is at the user’s 
//    own risk and responsibility.
//
// -------------------------------------------------------------------------
VAR_INPUT
  /// DetectionMode
  Value : DetectionMode;
END_VAR

CASE Value 
OF

  DetectionMode.TORQUE             : StrReplace('TORQUE ({0})'             ,'{0}' , USINT_TO_STRING(Value));
  DetectionMode.FORCE              : StrReplace('FORCE ({0})'              ,'{0}' , USINT_TO_STRING(Value));
  DetectionMode.ELECTRICAL_CURRENT : StrReplace('ELECTRICAL_CURRENT ({0})' ,'{0}' , USINT_TO_STRING(Value));
  DetectionMode.FOLLOWING_ERROR    : StrReplace('FOLLOWING_ERROR ({0})'    ,'{0}' , USINT_TO_STRING(Value));

END_CASE

END_FUNCTION

// Library/Functions/Convert/TO_STRING/ERROR_REACTION_TO_STRING
FUNCTION ERROR_REACTION_TO_STRING : STRING
// ------------------------------------------------------------------------- 
//  SRCI Robot Library                                                
// ------------------------------------------------------------------------- 
//                                                                           
//  Object:      ERROR_REACTION_TO_STRING                                       
//  Author:      Thorsten Brach                                                
//  Date:        2025-02-01
//
//  Description:                                              
//   
//                                                                           
//  Copyright: 
//    (C) 2025 Thorsten Brach. All rights reserved                                                                                                                                            
//             Licensed under the LGPL-3.0 license.
//                                                                           
//  Disclaimer:                                                                           
//    This project is provided without any guarantee and can be used for   
//    private and commercial purposes. Any use is at the user’s 
//    own risk and responsibility.
//
// -------------------------------------------------------------------------
VAR_INPUT
  /// ErrorReaction
  Value : ErrorReaction;
END_VAR

CASE Value 
OF

  ErrorReaction.ABORT_AND_MOVE : StrReplace('ABORT_AND_MOVE ({0})','{0}' , USINT_TO_STRING(Value));
  ErrorReaction.ABORT          : StrReplace('ABORT ({0})'         ,'{0}' , USINT_TO_STRING(Value));
  ErrorReaction.NO_REACTION    : StrReplace('NO_REACTION ({0})'   ,'{0}' , USINT_TO_STRING(Value));

END_CASE

END_FUNCTION

// Library/Functions/Convert/TO_STRING/ERROR_TRIGGER_MODE_TO_STRING
FUNCTION ERROR_TRIGGER_MODE_TO_STRING : STRING
// ------------------------------------------------------------------------- 
//  SRCI Robot Library                                                
// ------------------------------------------------------------------------- 
//                                                                           
//  Object:      ERROR_TRIGGER_MODE_TO_STRING                                       
//  Author:      Thorsten Brach                                                
//  Date:        2025-02-01
//
//  Description:                                              
//   
//                                                                           
//  Copyright: 
//    (C) 2025 Thorsten Brach. All rights reserved                                                                                                                                            
//             Licensed under the LGPL-3.0 license.
//                                                                           
//  Disclaimer:                                                                           
//    This project is provided without any guarantee and can be used for   
//    private and commercial purposes. Any use is at the user’s 
//    own risk and responsibility.
//
// -------------------------------------------------------------------------
VAR_INPUT
  /// ErrorTriggerMode
  Value : ErrorTriggerMode;
END_VAR

CASE Value 
OF

  ErrorTriggerMode.ANY_COMMAND                    : StrReplace('ANY_COMMAND ({0})'                    ,'{0}' , SINT_TO_STRING(Value));
  ErrorTriggerMode.GENERAL_COMMANDS               : StrReplace('GENERAL_COMMANDS ({0})'               ,'{0}' , SINT_TO_STRING(Value));
  ErrorTriggerMode.ADMINISTRATIVE_COMMANDS        : StrReplace('ADMINISTRATIVE_COMMANDS ({0})'        ,'{0}' , SINT_TO_STRING(Value));
  ErrorTriggerMode.MOVE_COMMANDS                  : StrReplace('MOVE_COMMANDS ({0})'                  ,'{0}' , SINT_TO_STRING(Value));
  ErrorTriggerMode.PERIPHERY_COMMANDS             : StrReplace('PERIPHERY_COMMANDS ({0})'             ,'{0}' , SINT_TO_STRING(Value));
  ErrorTriggerMode.EXTENDED_COMMANDS              : StrReplace('EXTENDED_COMMANDS ({0})'              ,'{0}' , SINT_TO_STRING(Value));
  ErrorTriggerMode.SPECIFIC_COMMAND_OR_RI_MESSAGE : StrReplace('SPECIFIC_COMMAND_OR_RI_MESSAGE ({0})' ,'{0}' , SINT_TO_STRING(Value));
  ErrorTriggerMode.SPECIFIC_RC_OR_RA_MESSAGE_CODE : StrReplace('SPECIFIC_RC_OR_RA_MESSAGE_CODE ({0})' ,'{0}' , SINT_TO_STRING(Value));
  ErrorTriggerMode.ANY_RI_MESSAGE_CODE            : StrReplace('ANY_RI_MESSAGE_CODE ({0})'            ,'{0}' , SINT_TO_STRING(Value));
  ErrorTriggerMode.ANY_RC_OR_RA_MESSAGE_CODE      : StrReplace('ANY_RC_OR_RA_MESSAGE_CODE ({0})'      ,'{0}' , SINT_TO_STRING(Value));

END_CASE

END_FUNCTION

// Library/Functions/Convert/TO_STRING/EXECUTION_MODE_TO_STRING
FUNCTION EXECUTION_MODE_TO_STRING : STRING
// ------------------------------------------------------------------------- 
//  SRCI Robot Library                                                
// ------------------------------------------------------------------------- 
//                                                                           
//  Object:      EXECUTION_MODE_TO_STRING                                       
//  Author:      Thorsten Brach                                                
//  Date:        2025-01-20
//
//  Description:                                              
//   
//                                                                           
//  Copyright: 
//    (C) 2024 Thorsten Brach. All rights reserved                                                                                                                                            
//             Licensed under the LGPL-3.0 license.
//                                                                           
//  Disclaimer:                                                                           
//    This project is provided without any guarantee and can be used for   
//    private and commercial purposes. Any use is at the user’s 
//    own risk and responsibility.
//
// -------------------------------------------------------------------------
VAR_INPUT
  /// ExecMode
  Value : ExecutionMode;
END_VAR

CASE Value
OF
  ExecutionMode.SEQUENCE_PRIMARY                 : EXECUTION_MODE_TO_STRING := StrReplace('SEQUENCE_PRIMARY ({0})'                 ,'{0}', USINT_TO_STRING(Value));
  ExecutionMode.SEQUENCE_ABORT_OTHERS_PRIMARY    : EXECUTION_MODE_TO_STRING := StrReplace('SEQUENCE_ABORT_OTHERS_PRIMARY ({0})'    ,'{0}', USINT_TO_STRING(Value));
  ExecutionMode.PARALLEL                         : EXECUTION_MODE_TO_STRING := StrReplace('PARALLEL ({0})'                         ,'{0}', USINT_TO_STRING(Value));
  ExecutionMode.CONTINUOUS                       : EXECUTION_MODE_TO_STRING := StrReplace('CONTINUOUS ({0})'                       ,'{0}', USINT_TO_STRING(Value));
  ExecutionMode.TRIGGER_MULTIPLE                 : EXECUTION_MODE_TO_STRING := StrReplace('TRIGGER_MULTIPLE ({0})'                 ,'{0}', USINT_TO_STRING(Value));
  ExecutionMode.SEQUENCE_SECONDARY               : EXECUTION_MODE_TO_STRING := StrReplace('SEQUENCE_SECONDARY ({0})'               ,'{0}', USINT_TO_STRING(Value));
  ExecutionMode.SEQUENCE_ABORT_OTHERS_SECONDARY  : EXECUTION_MODE_TO_STRING := StrReplace('SEQUENCE_ABORT_OTHERS_SECONDARY ({0})'  ,'{0}', USINT_TO_STRING(Value));
  ExecutionMode.STOP_PARALLEL_CONTINUOUS_TRIGGER : EXECUTION_MODE_TO_STRING := StrReplace('STOP_PARALLEL_CONTINUOUS_TRIGGER ({0})' ,'{0}', USINT_TO_STRING(Value));
ELSE
  EXECUTION_MODE_TO_STRING := 'UNKNOWN';
END_CASE

END_FUNCTION

// Library/Functions/Convert/TO_STRING/FRAGMENT_ACTION_TO_STRING
FUNCTION FRAGMENT_ACTION_TO_STRING : STRING
// ------------------------------------------------------------------------- 
//  SRCI Robot Library                                                
// ------------------------------------------------------------------------- 
//                                                                           
//  Object:      FRAGMENT_ACTION_TO_STRING                                       
//  Author:      Thorsten Brach                                                
//  Date:        2024-11-16
//
//  Description:                                              
//   
//                                                                           
//  Copyright: 
//    (C) 2024 Thorsten Brach. All rights reserved                                                                                                                                            
//             Licensed under the LGPL-3.0 license.
//                                                                           
//  Disclaimer:                                                                           
//    This project is provided without any guarantee and can be used for   
//    private and commercial purposes. Any use is at the user’s 
//    own risk and responsibility.
//
// -------------------------------------------------------------------------
VAR_INPUT
  /// Fragment action
  FragmentAction : BYTE;
END_VAR

IF ( FragmentAction.0 )
THEN
 FRAGMENT_ACTION_TO_STRING := CONCAT(FRAGMENT_ACTION_TO_STRING, ' Complete (Bit 0)');
END_IF

IF ( FragmentAction.1 )
THEN
 FRAGMENT_ACTION_TO_STRING := CONCAT(FRAGMENT_ACTION_TO_STRING, ' Reset (Bit 1)');
END_IF

IF ( FragmentAction.2 )
THEN
 FRAGMENT_ACTION_TO_STRING := CONCAT(FRAGMENT_ACTION_TO_STRING, ' Clear (Bit 2)');
END_IF

END_FUNCTION

// Library/Functions/Convert/TO_STRING/FRAME_CALCULATION_MODE_TO_STRING
FUNCTION FRAME_CALCULATION_MODE_TO_STRING : STRING
// ------------------------------------------------------------------------- 
//  SRCI Robot Library                                                
// ------------------------------------------------------------------------- 
//                                                                           
//  Object:      FRAME_CALCULATION_MODE_TO_STRING                                       
//  Author:      Thorsten Brach                                                
//  Date:        2025-02-01
//
//  Description:                                              
//   
//                                                                           
//  Copyright: 
//    (C) 2025 Thorsten Brach. All rights reserved                                                                                                                                            
//             Licensed under the LGPL-3.0 license.
//                                                                           
//  Disclaimer:                                                                           
//    This project is provided without any guarantee and can be used for   
//    private and commercial purposes. Any use is at the user’s 
//    own risk and responsibility.
//
// -------------------------------------------------------------------------
VAR_INPUT
  /// FrameCalculationMode
  Value : FrameCalculationMode;
END_VAR

CASE Value 
OF

  FrameCalculationMode.THREE_POINT_METHOD : StrReplace('THREE_POINT_METHOD ({0})','{0}' , SINT_TO_STRING(Value));
  FrameCalculationMode.FOUR_POINT_METHOD  : StrReplace('FOUR_POINT_METHOD ({0})' ,'{0}' , SINT_TO_STRING(Value));
  FrameCalculationMode.ONE_POINT_METHOD   : StrReplace('ONE_POINT_METHOD ({0})'  ,'{0}' , SINT_TO_STRING(Value));

END_CASE

END_FUNCTION

// Library/Functions/Convert/TO_STRING/IEC_DATE_TO_STRING
FUNCTION IEC_DATE_TO_STRING : STRING
// ------------------------------------------------------------------------- 
//  SRCI Robot Library                                                
// ------------------------------------------------------------------------- 
//                                                                           
//  Object:      IEC_DATE_TO_STRING                                       
//  Author:      Thorsten Brach                                                
//  Date:        2025-02-01
//
//  Description:                                              
//   
//                                                                           
//  Copyright: 
//    (C) 2025 Thorsten Brach. All rights reserved                                                                                                                                            
//             Licensed under the LGPL-3.0 license.
//                                                                           
//  Disclaimer:                                                                           
//    This project is provided without any guarantee and can be used for   
//    private and commercial purposes. Any use is at the user’s 
//    own risk and responsibility.
//
// -------------------------------------------------------------------------
VAR_INPUT
  /// IEC Date
  Value : IEC_DATE;
END_VAR

VAR
  /// temporary date
 _tmpData : DATE;
END_VAR

IEC_DATE_TO_STRING := DATE_TO_STRING(IEC_DATE_TO_DATE(Value));

END_FUNCTION

// Library/Functions/Convert/TO_STRING/IEC_TIME_TO_STRING
FUNCTION IEC_TIME_TO_STRING : STRING
// ------------------------------------------------------------------------- 
//  SRCI Robot Library                                                
// ------------------------------------------------------------------------- 
//                                                                           
//  Object:      ORI_MODE_TO_STRING                                       
//  Author:      Thorsten Brach                                                
//  Date:        2025-01-24
//
//  Description:                                              
//   
//                                                                           
//  Copyright: 
//    (C) 2025 Thorsten Brach. All rights reserved                                                                                                                                            
//             Licensed under the LGPL-3.0 license.
//                                                                           
//  Disclaimer:                                                                           
//    This project is provided without any guarantee and can be used for   
//    private and commercial purposes. Any use is at the user’s 
//    own risk and responsibility.
//
// -------------------------------------------------------------------------
VAR_INPUT
  /// IEC_TIME
  Value : IEC_TIME;
END_VAR
VAR
  /// temporary date
 _tmpData : DATE;
END_VAR

IEC_TIME_TO_STRING := TOD_TO_STRING(IEC_TIME_TO_TIME(Value));

END_FUNCTION

// Library/Functions/Convert/TO_STRING/ORI_MODE_TO_STRING
FUNCTION ORI_MODE_TO_STRING : STRING
// ------------------------------------------------------------------------- 
//  SRCI Robot Library                                                
// ------------------------------------------------------------------------- 
//                                                                           
//  Object:      ORI_MODE_TO_STRING                                       
//  Author:      Thorsten Brach                                                
//  Date:        2025-01-24
//
//  Description:                                              
//   
//                                                                           
//  Copyright: 
//    (C) 2025 Thorsten Brach. All rights reserved                                                                                                                                            
//             Licensed under the LGPL-3.0 license.
//                                                                           
//  Disclaimer:                                                                           
//    This project is provided without any guarantee and can be used for   
//    private and commercial purposes. Any use is at the user’s 
//    own risk and responsibility.
//
// -------------------------------------------------------------------------
VAR_INPUT
  /// OriMode
  Value : OriMode;
END_VAR

CASE Value 
OF

  OriMode.LINEAR_INTERPOLATED : StrReplace('LINEAR_INTERPOLATED ({0})','{0}' , USINT_TO_STRING(Value));
  OriMode.JOINT_INTERPOLATED  : StrReplace('JOINT_INTERPOLATED ({0})' ,'{0}' , USINT_TO_STRING(Value));
  OriMode.FIX                 : StrReplace('FIX ({0})'                ,'{0}' , USINT_TO_STRING(Value));
  OriMode.PATH                : StrReplace('PATH ({0})'               ,'{0}' , USINT_TO_STRING(Value));

END_CASE

END_FUNCTION

// Library/Functions/Convert/TO_STRING/INTERPOLATION_MODE_TO_STRING
FUNCTION INTERPOLATION_MODE_TO_STRING : STRING
// ------------------------------------------------------------------------- 
//  SRCI Robot Library                                                
// ------------------------------------------------------------------------- 
//                                                                           
//  Object:      INTERPOLATION_MODE_TO_STRING                                       
//  Author:      Thorsten Brach                                                
//  Date:        2025-02-01
//
//  Description:                                              
//   
//                                                                           
//  Copyright: 
//    (C) 2025 Thorsten Brach. All rights reserved                                                                                                                                            
//             Licensed under the LGPL-3.0 license.
//                                                                           
//  Disclaimer:                                                                           
//    This project is provided without any guarantee and can be used for   
//    private and commercial purposes. Any use is at the user’s 
//    own risk and responsibility.
//
// -------------------------------------------------------------------------
VAR_INPUT
  /// InterpolationMode
  Value : InterpolationMode;
END_VAR

CASE Value 
OF

  InterpolationMode.LINEAR_INTERPOLATION : StrReplace('LINEAR_INTERPOLATION ({0})' ,'{0}' , USINT_TO_STRING(Value));
  InterpolationMode.DIRECT_INTERPOLATION : StrReplace('DIRECT_INTERPOLATION ({0})' ,'{0}' , USINT_TO_STRING(Value));

END_CASE

END_FUNCTION

// Library/Functions/Convert/TO_STRING/JOG_MODE_TO_STRING
FUNCTION JOG_MODE_TO_STRING : STRING
// ------------------------------------------------------------------------- 
//  SRCI Robot Library                                                
// ------------------------------------------------------------------------- 
//                                                                           
//  Object:      JOG_MODE_TO_STRING                                       
//  Author:      Thorsten Brach                                                
//  Date:        2025-01-20
//
//  Description:                                              
//   
//                                                                           
//  Copyright: 
//    (C) 2025 Thorsten Brach. All rights reserved                                                                                                                                            
//             Licensed under the LGPL-3.0 license.
//                                                                           
//  Disclaimer:                                                                           
//    This project is provided without any guarantee and can be used for   
//    private and commercial purposes. Any use is at the user’s 
//    own risk and responsibility.
//
// -------------------------------------------------------------------------
VAR_INPUT
  /// JogMode
  Value : JogMode;
END_VAR

CASE Value 
OF
  
  JogMode.JOG_FRAME : JOG_MODE_TO_STRING := StrReplace('JOG_FRAME ({0})','{0}' , USINT_TO_STRING(Value));
  JogMode.JOG_TOOL  : JOG_MODE_TO_STRING := StrReplace('JOG_TOOL ({0})','{0}'  , USINT_TO_STRING(Value));
  JogMode.JOG_AXES  : JOG_MODE_TO_STRING := StrReplace('JOG_AXES ({0})','{0}'  , USINT_TO_STRING(Value));

END_CASE

END_FUNCTION

// Library/Functions/Convert/TO_STRING/LIMIT_MODE_TO_STRING
FUNCTION LIMIT_MODE_TO_STRING : STRING
// ------------------------------------------------------------------------- 
//  SRCI Robot Library                                                
// ------------------------------------------------------------------------- 
//                                                                           
//  Object:      LIMIT_MODE_TO_STRING                                       
//  Author:      Thorsten Brach                                                
//  Date:        2025-01-24
//
//  Description:                                              
//   
//                                                                           
//  Copyright: 
//    (C) 2025 Thorsten Brach. All rights reserved                                                                                                                                            
//             Licensed under the LGPL-3.0 license.
//                                                                           
//  Disclaimer:                                                                           
//    This project is provided without any guarantee and can be used for   
//    private and commercial purposes. Any use is at the user’s 
//    own risk and responsibility.
//
// -------------------------------------------------------------------------
VAR_INPUT
  /// LimitMode
  Value : LimitMode;
END_VAR

CASE Value 
OF

  LimitMode.LIMIT_DEFINED    : StrReplace('LIMIT_DEFINED ({0})'    ,'{0}' , USINT_TO_STRING(Value));
  LimitMode.NO_LIMIT_DEFINED : StrReplace('NO_LIMIT_DEFINED ({0})' ,'{0}' , USINT_TO_STRING(Value));

END_CASE

END_FUNCTION

// Library/Functions/Convert/TO_STRING/LOAD_MEASUREMENT_MODE_TO_STRING
FUNCTION LOAD_MEASUREMENT_MODE_TO_STRING : STRING
// ------------------------------------------------------------------------- 
//  SRCI Robot Library                                                
// ------------------------------------------------------------------------- 
//                                                                           
//  Object:      LOAD_MEASUREMENT_MODE_TO_STRING                                       
//  Author:      Thorsten Brach                                                
//  Date:        2025-02-01
//
//  Description:                                              
//   
//                                                                           
//  Copyright: 
//    (C) 2025 Thorsten Brach. All rights reserved                                                                                                                                            
//             Licensed under the LGPL-3.0 license.
//                                                                           
//  Disclaimer:                                                                           
//    This project is provided without any guarantee and can be used for   
//    private and commercial purposes. Any use is at the user’s 
//    own risk and responsibility.
//
// -------------------------------------------------------------------------
VAR_INPUT
  /// LoadMeasurementMode
  Value : LoadMeasurementMode;
END_VAR

CASE Value 
OF

  LoadMeasurementMode.ONE_POSITION         : StrReplace('ONE_POSITION ({0})'        ,'{0}' , USINT_TO_STRING(Value));
  LoadMeasurementMode.CONFIGURATION_ANGLE  : StrReplace('CONFIGURATION_ANGLE ({0})' ,'{0}' , USINT_TO_STRING(Value));
  LoadMeasurementMode.AREA                 : StrReplace('AREA ({0})'                ,'{0}' , USINT_TO_STRING(Value));
  LoadMeasurementMode.TWO_POSITIONS        : StrReplace('TWO_POSITIONS ({0})'       ,'{0}' , USINT_TO_STRING(Value));

END_CASE

END_FUNCTION

// Library/Functions/Convert/TO_STRING/LOAD_MEASUREMENT_STEPS_TO_STRING
FUNCTION LOAD_MEASUREMENT_STEPS_TO_STRING : STRING
// ------------------------------------------------------------------------- 
//  SRCI Robot Library                                                
// ------------------------------------------------------------------------- 
//                                                                           
//  Object:      LOAD_MEASUREMENT_STEPS_TO_STRING                                       
//  Author:      Thorsten Brach                                                
//  Date:        2025-02-01
//
//  Description:                                              
//   
//                                                                           
//  Copyright: 
//    (C) 2025 Thorsten Brach. All rights reserved                                                                                                                                            
//             Licensed under the LGPL-3.0 license.
//                                                                           
//  Disclaimer:                                                                           
//    This project is provided without any guarantee and can be used for   
//    private and commercial purposes. Any use is at the user’s 
//    own risk and responsibility.
//
// -------------------------------------------------------------------------
VAR_INPUT
  /// LoadMeasurementSteps
  Value : LoadMeasurementSteps;
END_VAR

CASE Value 
OF

  LoadMeasurementSteps.RESET            : StrReplace('RESET ({0})'            ,'{0}' , USINT_TO_STRING(Value));
  LoadMeasurementSteps.FIRST_POSITION   : StrReplace('FIRST_POSITION ({0})'   ,'{0}' , USINT_TO_STRING(Value));
  LoadMeasurementSteps.SECOND_POSITION  : StrReplace('SECOND_POSITION ({0})'  ,'{0}' , USINT_TO_STRING(Value));
  LoadMeasurementSteps.THIRD_POSITION   : StrReplace('THIRD_POSITION ({0})'   ,'{0}' , USINT_TO_STRING(Value));
  LoadMeasurementSteps.FOURTH_POSITION  : StrReplace('FOURTH_POSITION ({0})'  ,'{0}' , USINT_TO_STRING(Value));
  LoadMeasurementSteps.LOAD_CALCULATION : StrReplace('LOAD_CALCULATION ({0})' ,'{0}' , USINT_TO_STRING(Value));
  
END_CASE

END_FUNCTION

// Library/Functions/Convert/TO_STRING/LOG_LEVEL_TO_STRING
FUNCTION LOG_LEVEL_TO_STRING : STRING
// ------------------------------------------------------------------------- 
//  SRCI Robot Library                                                
// ------------------------------------------------------------------------- 
//                                                                           
//  Object:      LOG_LEVEL_TO_STRING                                       
//  Author:      Thorsten Brach                                                
//  Date:        2025-01-24
//
//  Description:                                              
//   
//                                                                           
//  Copyright: 
//    (C) 2025 Thorsten Brach. All rights reserved                                                                                                                                            
//             Licensed under the LGPL-3.0 license.
//                                                                           
//  Disclaimer:                                                                           
//    This project is provided without any guarantee and can be used for   
//    private and commercial purposes. Any use is at the user’s 
//    own risk and responsibility.
//
// -------------------------------------------------------------------------
VAR_INPUT
  /// LogLevel
  Value : LogLevel;
END_VAR

CASE Value 
OF

  LogLevel.DEACTIVATE  : StrReplace('DEACTIVATE ({0})' ,'{0}' , SINT_TO_STRING(Value));
  LogLevel.DEBUG       : StrReplace('DEBUG ({0})'      ,'{0}' , SINT_TO_STRING(Value));
  LogLevel.INFO        : StrReplace('INFO ({0})'       ,'{0}' , SINT_TO_STRING(Value));
  LogLevel.WARNING     : StrReplace('WARNING ({0})'    ,'{0}' , SINT_TO_STRING(Value));
  LogLevel.ERROR       : StrReplace('ERROR ({0})'      ,'{0}' , SINT_TO_STRING(Value));
  LogLevel.FATAL_ERROR : StrReplace('FATAL_ERROR ({0})','{0}' , SINT_TO_STRING(Value));

END_CASE

END_FUNCTION

// Library/Functions/Convert/TO_STRING/LOGON_MODE_TO_STRING
FUNCTION LOGON_MODE_TO_STRING : STRING
// ------------------------------------------------------------------------- 
//  SRCI Robot Library                                                
// ------------------------------------------------------------------------- 
//                                                                           
//  Object:      LOGON_MODE_TO_STRING                                       
//  Author:      Thorsten Brach                                                
//  Date:        2025-02-01
//
//  Description:                                              
//   
//                                                                           
//  Copyright: 
//    (C) 2025 Thorsten Brach. All rights reserved                                                                                                                                            
//             Licensed under the LGPL-3.0 license.
//                                                                           
//  Disclaimer:                                                                           
//    This project is provided without any guarantee and can be used for   
//    private and commercial purposes. Any use is at the user’s 
//    own risk and responsibility.
//
// -------------------------------------------------------------------------
VAR_INPUT
  /// LogonMode
  Value : LogonMode;
END_VAR

CASE Value 
OF

  LogonMode.PASSWORD_ONLY         : StrReplace('PASSWORD_ONLY ({0})'         ,'{0}' , SINT_TO_STRING(Value));
  LogonMode.USERNAME_AND_PASSWORD : StrReplace('USERNAME_AND_PASSWORD ({0})' ,'{0}' , SINT_TO_STRING(Value));
  LogonMode.LEVEL_ID_AND_PASSWORD : StrReplace('LEVEL_ID_AND_PASSWORD ({0})' ,'{0}' , SINT_TO_STRING(Value));

END_CASE

END_FUNCTION

// Library/Functions/Convert/TO_STRING/MEASUREING_UNIT_MODE_TO_STRING
FUNCTION MEASUREING_UNIT_MODE_TO_STRING : STRING
// ------------------------------------------------------------------------- 
//  SRCI Robot Library                                                
// ------------------------------------------------------------------------- 
//                                                                           
//  Object:      MEASUREING_UNIT_MODE_TO_STRING                                       
//  Author:      Thorsten Brach                                                
//  Date:        2025-01-24
//
//  Description:                                              
//   
//                                                                           
//  Copyright: 
//    (C) 2025 Thorsten Brach. All rights reserved                                                                                                                                            
//             Licensed under the LGPL-3.0 license.
//                                                                           
//  Disclaimer:                                                                           
//    This project is provided without any guarantee and can be used for   
//    private and commercial purposes. Any use is at the user’s 
//    own risk and responsibility.
//
// -------------------------------------------------------------------------
VAR_INPUT
  /// MeasuringUnitMode
  Value : MeasuringUnitMode;
END_VAR

CASE Value 
OF

  MeasuringUnitMode.VECTOR_LENGTH  : StrReplace('VECTOR_LENGTH ({0})'  ,'{0}' , USINT_TO_STRING(Value));
  MeasuringUnitMode.SEGMENT_LENGTH : StrReplace('SEGMENT_LENGTH ({0})' ,'{0}' , USINT_TO_STRING(Value));
  MeasuringUnitMode.TIME_DURATION  : StrReplace('TIME_DURATION ({0})'  ,'{0}' , USINT_TO_STRING(Value));

END_CASE

END_FUNCTION

// Library/Functions/Convert/TO_STRING/MESSAGE_TYPE_TO_STRING
FUNCTION MESSAGE_TYPE_TO_STRING : STRING
// ------------------------------------------------------------------------- 
//  SRCI Robot Library                                                
// ------------------------------------------------------------------------- 
//                                                                           
//  Object:      MESSAGE_TYPE_TO_STRING                                       
//  Author:      Thorsten Brach                                                
//  Date:        2025-01-11
//
//  Description:                                              
//   
//                                                                           
//  Copyright: 
//    (C) 2025 Thorsten Brach. All rights reserved                                                                                                                                            
//             Licensed under the LGPL-3.0 license.
//                                                                           
//  Disclaimer:                                                                           
//    This project is provided without any guarantee and can be used for   
//    private and commercial purposes. Any use is at the user’s 
//    own risk and responsibility.
//
// -------------------------------------------------------------------------
VAR_INPUT
  /// Severity
  Value     : MessageType;
  /// Fill spaces to the end, so that all values has the same length  
  AlignString : BOOL;
END_VAR

IF (AlignString)
THEN
  CASE Value OF
    
    MessageType.RI  : MESSAGE_TYPE_TO_STRING := 'RI ';
    MessageType.RC  : MESSAGE_TYPE_TO_STRING := 'RC ';
    MessageType.RA  : MESSAGE_TYPE_TO_STRING := 'RA ';
    MessageType.CMD : MESSAGE_TYPE_TO_STRING := 'CMD' ;
  ELSE
    MESSAGE_TYPE_TO_STRING := '???'; 
  END_CASE
ELSE
  CASE Value OF
    
    MessageType.RI  : MESSAGE_TYPE_TO_STRING := 'RI';
    MessageType.RC  : MESSAGE_TYPE_TO_STRING := 'RC';
    MessageType.RA  : MESSAGE_TYPE_TO_STRING := 'RA';
    MessageType.CMD : MESSAGE_TYPE_TO_STRING := 'CMD' ;
  ELSE
    MESSAGE_TYPE_TO_STRING := '???'; 
  END_CASE  
END_IF

END_FUNCTION

// Library/Functions/Convert/TO_STRING/REFERENCE_TYPE_TO_STRING
FUNCTION REFERENCE_TYPE_TO_STRING : STRING
// ------------------------------------------------------------------------- 
//  SRCI Robot Library                                                
// ------------------------------------------------------------------------- 
//                                                                           
//  Object:      REFERENCE_TYPE_TO_STRING                                       
//  Author:      Thorsten Brach                                                
//  Date:        2025-01-24
//
//  Description:                                              
//   
//                                                                           
//  Copyright: 
//    (C) 2025 Thorsten Brach. All rights reserved                                                                                                                                            
//             Licensed under the LGPL-3.0 license.
//                                                                           
//  Disclaimer:                                                                           
//    This project is provided without any guarantee and can be used for   
//    private and commercial purposes. Any use is at the user’s 
//    own risk and responsibility.
//
// -------------------------------------------------------------------------
VAR_INPUT
  /// ReferenceType
  Value : ReferenceType;
END_VAR

CASE Value 
OF

  ReferenceType.TOOL  : StrReplace('TOOL ({0})'  ,'{0}' , USINT_TO_STRING(Value));
  ReferenceType.FRAME : StrReplace('FRAME ({0})' ,'{0}' , USINT_TO_STRING(Value));

END_CASE

END_FUNCTION

// Library/Functions/Convert/TO_STRING/SENSOR_CONNECTION_MODE_TO_STRING
FUNCTION SENSOR_CONNECTION_MODE_TO_STRING : STRING
// ------------------------------------------------------------------------- 
//  SRCI Robot Library                                                
// ------------------------------------------------------------------------- 
//                                                                           
//  Object:      SENSOR_CONNECTION_MODE_TO_STRING                                       
//  Author:      Thorsten Brach                                                
//  Date:        2025-02-01
//
//  Description:                                              
//   
//                                                                           
//  Copyright: 
//    (C) 2025 Thorsten Brach. All rights reserved                                                                                                                                            
//             Licensed under the LGPL-3.0 license.
//                                                                           
//  Disclaimer:                                                                           
//    This project is provided without any guarantee and can be used for   
//    private and commercial purposes. Any use is at the user’s 
//    own risk and responsibility.
//
// -------------------------------------------------------------------------
VAR_INPUT
  /// SensorConnectionMode
  Value : SensorConnectionMode;
END_VAR

CASE Value 
OF

  SensorConnectionMode.RC_SENSOR_ALGORITHM     : StrReplace('RC_SENSOR_ALGORITHM ({0})'     ,'{0}' , USINT_TO_STRING(Value));
  SensorConnectionMode.PLC_SENSOR_RC_ALGORITHM : StrReplace('PLC_SENSOR_RC_ALGORITHM ({0})' ,'{0}' , USINT_TO_STRING(Value));
  SensorConnectionMode.PLC_SENSOR_ALGORITHM    : StrReplace('PLC_SENSOR_ALGORITHM ({0})'    ,'{0}' , USINT_TO_STRING(Value));

END_CASE

END_FUNCTION

// Library/Functions/Convert/TO_STRING/SEVERITY_TO_STRING
FUNCTION SEVERITY_TO_STRING : STRING
// ------------------------------------------------------------------------- 
//  SRCI Robot Library                                                
// ------------------------------------------------------------------------- 
//                                                                           
//  Object:      SEVERITY_TO_STRING                                       
//  Author:      Thorsten Brach                                                
//  Date:        2025-01-11
//
//  Description:                                              
//   
//                                                                           
//  Copyright: 
//    (C) 2025 Thorsten Brach. All rights reserved                                                                                                                                            
//             Licensed under the LGPL-3.0 license.
//                                                                           
//  Disclaimer:                                                                           
//    This project is provided without any guarantee and can be used for   
//    private and commercial purposes. Any use is at the user’s 
//    own risk and responsibility.
//
// -------------------------------------------------------------------------
VAR_INPUT
  /// Severity
  Value : Severity;
  /// Fill spaces to the end, so that all values has the same length  
  AlignString : BOOL;
END_VAR

IF (AlignString)
THEN
  CASE Value OF
    Severity.DEBUG       : SEVERITY_TO_STRING := 'DEBUG      ';
    Severity.INFO        : SEVERITY_TO_STRING := 'INFO       ';
    Severity.WARNING     : SEVERITY_TO_STRING := 'WARNING    ';
    Severity.ERROR       : SEVERITY_TO_STRING := 'ERROR      ' ;
    Severity.FATAL_ERROR : SEVERITY_TO_STRING := 'FATAL_ERROR' ;
  ELSE
    SEVERITY_TO_STRING := 'UNKOWN     '; 
  END_CASE
ELSE
  CASE Value OF
    Severity.DEBUG       : SEVERITY_TO_STRING := 'DEBUG';
    Severity.INFO        : SEVERITY_TO_STRING := 'INFO';
    Severity.WARNING     : SEVERITY_TO_STRING := 'WARNING';
    Severity.ERROR       : SEVERITY_TO_STRING := 'ERROR' ;
    Severity.FATAL_ERROR : SEVERITY_TO_STRING := 'FATAL_ERROR' ;
  ELSE
    SEVERITY_TO_STRING := 'UNKOWN'; 
  END_CASE
END_IF

END_FUNCTION

// Library/Functions/Convert/TO_STRING/SINGULARITY_AVOIDANCE_MODE_TO_STRING
FUNCTION SINGULARITY_AVOIDANCE_MODE_TO_STRING : STRING
// ------------------------------------------------------------------------- 
//  SRCI Robot Library                                                
// ------------------------------------------------------------------------- 
//                                                                           
//  Object:      SINGULARITY_AVOIDANCE_MODE_TO_STRING                                       
//  Author:      Thorsten Brach                                                
//  Date:        2025-01-24
//
//  Description:                                              
//   
//                                                                           
//  Copyright: 
//    (C) 2025 Thorsten Brach. All rights reserved                                                                                                                                            
//             Licensed under the LGPL-3.0 license.
//                                                                           
//  Disclaimer:                                                                           
//    This project is provided without any guarantee and can be used for   
//    private and commercial purposes. Any use is at the user’s 
//    own risk and responsibility.
//
// -------------------------------------------------------------------------
VAR_INPUT
  /// SingularityAvoidanceMode
  Value : SingularityAvoidanceMode;
END_VAR

CASE Value 
OF

  SingularityAvoidanceMode.NO_CHANGE        : StrReplace('NO_CHANGE ({0})'        ,'{0}' , USINT_TO_STRING(Value));
  SingularityAvoidanceMode.LOCK_J4          : StrReplace('LOCK_J4 ({0})'          ,'{0}' , USINT_TO_STRING(Value));
  SingularityAvoidanceMode.TOOL_ORIENTATION : StrReplace('TOOL_ORIENTATION ({0})' ,'{0}' , USINT_TO_STRING(Value));

END_CASE

END_FUNCTION

// Library/Functions/Convert/TO_STRING/SPLINE_MODE_TO_STRING
FUNCTION SPLINE_MODE_TO_STRING : STRING
// ------------------------------------------------------------------------- 
//  SRCI Robot Library                                                
// ------------------------------------------------------------------------- 
//                                                                           
//  Object:      SPLINE_MODE_TO_STRING                                       
//  Author:      Thorsten Brach                                                
//  Date:        2025-02-01
//
//  Description:                                              
//   
//                                                                           
//  Copyright: 
//    (C) 2025 Thorsten Brach. All rights reserved                                                                                                                                            
//             Licensed under the LGPL-3.0 license.
//                                                                           
//  Disclaimer:                                                                           
//    This project is provided without any guarantee and can be used for   
//    private and commercial purposes. Any use is at the user’s 
//    own risk and responsibility.
//
// -------------------------------------------------------------------------
VAR_INPUT
  /// SplineMode
  Value : SplineMode;
END_VAR

CASE Value 
OF

  SplineMode.DISCRETE_POINTS      : StrReplace('DISCRETE_POINTS ({0})'      ,'{0}' , UINT_TO_STRING(Value));
  SplineMode.BEZIER_SPLINE        : StrReplace('BEZIER_SPLINE ({0})'        ,'{0}' , UINT_TO_STRING(Value));
  SplineMode.B_SPLINES            : StrReplace('B_SPLINES ({0})'            ,'{0}' , UINT_TO_STRING(Value));
  SplineMode.CUBIC_HERMITE_SPLINE : StrReplace('CUBIC_HERMITE_SPLINE ({0})' ,'{0}' , UINT_TO_STRING(Value));
  SplineMode.C_SPLINES            : StrReplace('C_SPLINES ({0})'            ,'{0}' , UINT_TO_STRING(Value));

END_CASE

END_FUNCTION

// Library/Functions/Convert/TO_STRING/STEP_MODE_TO_STRING
FUNCTION STEP_MODE_TO_STRING : STRING
// ------------------------------------------------------------------------- 
//  SRCI Robot Library                                                
// ------------------------------------------------------------------------- 
//                                                                           
//  Object:      STEP_MODE_TO_STRING                                       
//  Author:      Thorsten Brach                                                
//  Date:        2025-01-18
//
//  Description:                                              
//   
//                                                                           
//  Copyright: 
//    (C) 2025 Thorsten Brach. All rights reserved                                                                                                                                            
//             Licensed under the LGPL-3.0 license.
//                                                                           
//  Disclaimer:                                                                           
//    This project is provided without any guarantee and can be used for   
//    private and commercial purposes. Any use is at the user’s 
//    own risk and responsibility.
//
// -------------------------------------------------------------------------
VAR_INPUT
  /// StepMode
  Value : StepMode;
END_VAR

CASE Value 
OF
  
  StepMode.DEACTIVATE : StrReplace('DEACTIVATE ({0})' ,'{0}' , USINT_TO_STRING(Value));
  StepMode.BLENDING   : StrReplace('BLENDING ({0})'   ,'{0}' , USINT_TO_STRING(Value));
  StepMode.EXACT_STOP : StrReplace('EXACT_STOP ({0})' ,'{0}' , USINT_TO_STRING(Value));

END_CASE

END_FUNCTION

// Library/Functions/Convert/TO_STRING/STOP_MODE_TO_STRING
FUNCTION STOP_MODE_TO_STRING : STRING
// ------------------------------------------------------------------------- 
//  SRCI Robot Library                                                
// ------------------------------------------------------------------------- 
//                                                                           
//  Object:      STOP_MODE_TO_STRING                                       
//  Author:      Thorsten Brach                                                
//  Date:        2025-01-24
//
//  Description:                                              
//   
//                                                                           
//  Copyright: 
//    (C) 2025 Thorsten Brach. All rights reserved                                                                                                                                            
//             Licensed under the LGPL-3.0 license.
//                                                                           
//  Disclaimer:                                                                           
//    This project is provided without any guarantee and can be used for   
//    private and commercial purposes. Any use is at the user’s 
//    own risk and responsibility.
//
// -------------------------------------------------------------------------
VAR_INPUT
  /// StopMode
  Value : StopMode;
END_VAR

CASE Value 
OF

  StopMode.STOP_ALL_SUBPROGRAMS : StrReplace('STOP_ALL_SUBPROGRAMS ({0})','{0}' , USINT_TO_STRING(Value));
  StopMode.STOP_INSTANCE_ID     : StrReplace('STOP_INSTANCE_ID ({0})'    ,'{0}' , USINT_TO_STRING(Value));
  StopMode.STOP_JOB_ID          : StrReplace('STOP_JOB_ID ({0})'         ,'{0}' , USINT_TO_STRING(Value));

END_CASE

END_FUNCTION

// Library/Functions/Convert/TO_STRING/SYNC_IN_MODE_TO_STRING
FUNCTION SYNC_IN_MODE_TO_STRING : STRING
// ------------------------------------------------------------------------- 
//  SRCI Robot Library                                                
// ------------------------------------------------------------------------- 
//                                                                           
//  Object:      SYNC_IN_MODE_TO_STRING                                       
//  Author:      Thorsten Brach                                                
//  Date:        2025-02-01
//
//  Description:                                              
//   
//                                                                           
//  Copyright: 
//    (C) 2025 Thorsten Brach. All rights reserved                                                                                                                                            
//             Licensed under the LGPL-3.0 license.
//                                                                           
//  Disclaimer:                                                                           
//    This project is provided without any guarantee and can be used for   
//    private and commercial purposes. Any use is at the user’s 
//    own risk and responsibility.
//
// -------------------------------------------------------------------------
VAR_INPUT
  /// SyncInMode
  Value : SyncInMode;
END_VAR

CASE Value 
OF

  SyncInMode.IN_SYNC_IN_ZONE : StrReplace('IN_SYNC_IN_ZONE ({0})','{0}' , USINT_TO_STRING(Value));
  SyncInMode.AFTER_DISTANCE  : StrReplace('AFTER_DISTANCE ({0})' ,'{0}' , USINT_TO_STRING(Value));
  SyncInMode.AFTER_TIME      : StrReplace('AFTER_TIME ({0})'     ,'{0}' , USINT_TO_STRING(Value));
  SyncInMode.IMMEDIATELY     : StrReplace('IMMEDIATELY ({0})'    ,'{0}' , USINT_TO_STRING(Value));

END_CASE

END_FUNCTION

// Library/Functions/Convert/TO_STRING/SYNC_REACTION_TO_STRING
FUNCTION SYNC_REACTION_TO_STRING : STRING
// ------------------------------------------------------------------------- 
//  SRCI Robot Library                                                
// ------------------------------------------------------------------------- 
//                                                                           
//  Object:      SYNC_REACTION_TO_STRING                                       
//  Author:      Thorsten Brach                                                
//  Date:        2025-01-24
//
//  Description:                                              
//   
//                                                                           
//  Copyright: 
//    (C) 2025 Thorsten Brach. All rights reserved                                                                                                                                            
//             Licensed under the LGPL-3.0 license.
//                                                                           
//  Disclaimer:                                                                           
//    This project is provided without any guarantee and can be used for   
//    private and commercial purposes. Any use is at the user’s 
//    own risk and responsibility.
//
// -------------------------------------------------------------------------
VAR_INPUT
  /// SyncReaction
  Value : SyncReaction;
END_VAR

CASE Value 
OF

  SyncReaction.NO_REACTION     : StrReplace('NO_REACTION ({0})'     ,'{0}' , USINT_TO_STRING(Value));
  SyncReaction.REACTION_TYPE_1 : StrReplace('REACTION_TYPE_1 ({0})' ,'{0}' , USINT_TO_STRING(Value));
  SyncReaction.REACTION_TYPE_2 : StrReplace('REACTION_TYPE_2 ({0})' ,'{0}' , USINT_TO_STRING(Value));
  SyncReaction.REACTION_TYPE_3 : StrReplace('REACTION_TYPE_3 ({0})' ,'{0}' , USINT_TO_STRING(Value));

END_CASE

END_FUNCTION

// Library/Functions/Convert/TO_STRING/TELEGRAM_CONTROL_TO_STRING
FUNCTION TELEGRAM_CONTROL_TO_STRING : STRING
// ------------------------------------------------------------------------- 
//  SRCI Robot Library                                                
// ------------------------------------------------------------------------- 
//                                                                           
//  Object:      TELEGRAM_CONTROL_TO_STRING                                       
//  Author:      Thorsten Brach                                                
//  Date:        2024-11-16
//
//  Description:                                              
//   
//                                                                           
//  Copyright: 
//    (C) 2024 Thorsten Brach. All rights reserved                                                                                                                                            
//             Licensed under the LGPL-3.0 license.
//                                                                           
//  Disclaimer:                                                                           
//    This project is provided without any guarantee and can be used for   
//    private and commercial purposes. Any use is at the user’s 
//    own risk and responsibility.
//
// -------------------------------------------------------------------------
VAR_INPUT
  /// Telegram state
  Control : ControlHalfByte;
END_VAR

CASE Control OF
  ControlHalfByte.NONE         : TELEGRAM_CONTROL_TO_STRING := StrReplace('NONE ({0})'        ,'{0}', USINT_TO_STRING(Control));
  ControlHalfByte.INITIALIZE   : TELEGRAM_CONTROL_TO_STRING := StrReplace('INITIALIZE ({0})'  ,'{0}', USINT_TO_STRING(Control));
  ControlHalfByte.RESUME       : TELEGRAM_CONTROL_TO_STRING := StrReplace('RESUME ({0})'      ,'{0}', USINT_TO_STRING(Control));
  ControlHalfByte.RESET        : TELEGRAM_CONTROL_TO_STRING := StrReplace('RESET ({0})'       ,'{0}', USINT_TO_STRING(Control));
  ControlHalfByte.ACK_ERROR    : TELEGRAM_CONTROL_TO_STRING := StrReplace('ACK_ERROR ({0})'   ,'{0}', USINT_TO_STRING(Control));
  ControlHalfByte.CLIENT_ERROR : TELEGRAM_CONTROL_TO_STRING := StrReplace('CLIENT_ERROR ({0})','{0}', USINT_TO_STRING(Control));  
ELSE
  TELEGRAM_CONTROL_TO_STRING := CONCAT('TelegramControlToString-Function: Error -> no parsing for value ', BYTE_TO_STRING(Control));
END_CASE

END_FUNCTION

// Library/Functions/Convert/TO_STRING/TELEGRAM_STATE_TO_STRING
FUNCTION TELEGRAM_STATE_TO_STRING : STRING
// ------------------------------------------------------------------------- 
//  SRCI Robot Library                                                
// ------------------------------------------------------------------------- 
//                                                                           
//  Object:      TelegramStateToString                                       
//  Author:      Thorsten Brach                                                
//  Date:        2024-11-16
//
//  Description:                                              
//   
//                                                                           
//  Copyright: 
//    (C) 2024 Thorsten Brach. All rights reserved                                                                                                                                            
//             Licensed under the LGPL-3.0 license.
//                                                                           
//  Disclaimer:                                                                           
//    This project is provided without any guarantee and can be used for   
//    private and commercial purposes. Any use is at the user’s 
//    own risk and responsibility.
//
// -------------------------------------------------------------------------
VAR_INPUT
  /// Telegram state
  State : TelegramState;
END_VAR

CASE State OF

